FUNCTION_BLOCK PtTimeSource IMPLEMENTS I_PtTimesource
VAR_INPUT
END_VAR
VAR_OUTPUT
END_VAR
VAR
	_DateTime : ptDateTime;
	DefaultTimeZoneTime : TIMESTRUCT;
	
END_VAR

METHOD getDateTime : PtDateTime
VAR_INPUT
END_VAR

DefaultTimeZoneTime := FILETIME64_TO_SYSTEMTIME(fileTime:= F_GetSystemTime());
_DateTime.Set(
	Year:= DefaultTimeZoneTime.wYear, 
	Month:= DefaultTimeZoneTime.wMonth, 
	Day:= DefaultTimeZoneTime.wDay, 
	Hour:= DefaultTimeZoneTime.wHour, 
	Minute:= DefaultTimeZoneTime.wMinute, 
	Second:= DefaultTimeZoneTime.wSecond, 
	Microsecond:= DefaultTimeZoneTime.wMilliseconds, 
	TimeZone:= 0);
getDateTime := _DateTime;
END_METHOD

END_FUNCTION_BLOCK

(* stored: Version 1.1.0.1, ProductVersion 3.1.4024.12
   POU PtTimeSource: Id {7f86d321-e204-4b9b-8326-b9d9c83135d7}, SpecialFunc None
   Method getDateTime: Id {89201670-5233-43cd-af28-06268916d322} *)
